// TIA Portal V17 export
// export: Created 2025-03-07T09:17:48.5611962Z, ExportSetting WithDefaults, DisplayName Totally Integrated Automation Portal, DisplayVersion V17 Update 8, DisplayName TIA Portal Openness, DisplayVersion V17 Update 8, DisplayName TIA Portal Version Control Interface, DisplayVersion V17, DisplayName SINAMICS Startdrive Advanced, DisplayVersion V17 SP2, DisplayName SINAMICS Startdrive G110M, G120, G120C, G120D, G120P, G115D, DisplayVersion V17 SP2, DisplayName SINAMICS Startdrive G130, G150, S120, S150, SINAMICS MV, S210, DisplayVersion V17 SP2, DisplayName STEP 7 Professional, DisplayVersion V17 Update 8, DisplayName SINUMERIK ONE STEP 7 Toolbox, DisplayVersion V17 Update 12, DisplayName SINUMERIK 840D sl STEP 7 Toolbox, DisplayVersion V17 Update 12, DisplayName STEP 7 Safety, DisplayVersion V17 Update 6, DisplayName WinCC Advanced, DisplayVersion V17 Update 8
FUNCTION "FC2102_INFEED_MODULE" : Void   // FC2102, LAD
{ S7_Optimized_Access := 'FALSE' }
AUTHOR : ETXETAR
VERSION : 1.0
// stored: AutoNumber false, IsIECCheckEnabled false, SetENOAutomatically false, UDAEnableTagReadback false
   VAR_TEMP
      O_BYTE_0 : Struct   // OPTIONS BYTE 0
         POWER_SUPPLY_2 : Bool;   // POWER SUPPLY 2 OPTION
      END_STRUCT;
   END_VAR
   VAR CONSTANT
      FC_NUMBER : DInt := 2102;
   END_VAR
   VAR_TEMP   // added for the SCL form of the ladder/FBD networks
      _w1 : Bool;
   END_VAR
BEGIN

REGION Network 1: OPTIONS OFF
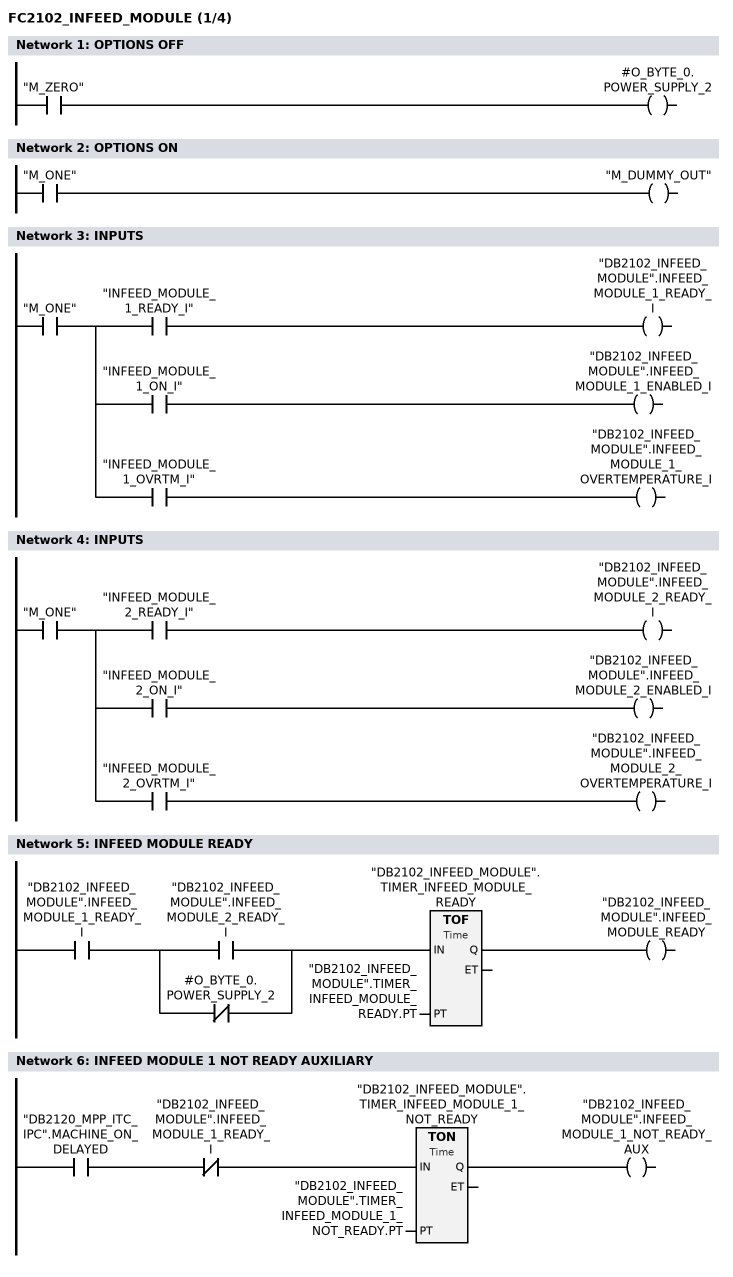
   RUNG wire#powerrail
      Contact( "M_ZERO" )
      Coil( #O_BYTE_0.POWER_SUPPLY_2 )
   END_RUNG
   // the same network as SCL:
   #O_BYTE_0.POWER_SUPPLY_2 := "M_ZERO";
END_REGION

REGION Network 2: OPTIONS ON
   RUNG wire#powerrail
      Contact( "M_ONE" )
      Coil( "M_DUMMY_OUT" )
   END_RUNG
   // the same network as SCL:
   "M_DUMMY_OUT" := "M_ONE";
END_REGION

REGION Network 3: INPUTS
   RUNG wire#powerrail
      Contact( "M_ONE" )
      wire#w1
      Contact( "INFEED_MODULE_1_READY_I" )
      Coil( "DB2102_INFEED_MODULE".INFEED_MODULE_1_READY_I )
   END_RUNG
   RUNG wire#w1
      Contact( "INFEED_MODULE_1_ON_I" )
      Coil( "DB2102_INFEED_MODULE".INFEED_MODULE_1_ENABLED_I )
   END_RUNG
   RUNG wire#w1
      Contact( "INFEED_MODULE_1_OVRTM_I" )
      Coil( "DB2102_INFEED_MODULE".INFEED_MODULE_1_OVERTEMPERATURE_I )
   END_RUNG
   // the same network as SCL:
   "DB2102_INFEED_MODULE".INFEED_MODULE_1_READY_I := "M_ONE" AND "INFEED_MODULE_1_READY_I";
   "DB2102_INFEED_MODULE".INFEED_MODULE_1_ENABLED_I := "M_ONE" AND "INFEED_MODULE_1_ON_I";
   "DB2102_INFEED_MODULE".INFEED_MODULE_1_OVERTEMPERATURE_I := "M_ONE" AND "INFEED_MODULE_1_OVRTM_I";
END_REGION

REGION Network 4: INPUTS
   RUNG wire#powerrail
      Contact( "M_ONE" )
      wire#w1
      Contact( "INFEED_MODULE_2_READY_I" )
      Coil( "DB2102_INFEED_MODULE".INFEED_MODULE_2_READY_I )
   END_RUNG
   RUNG wire#w1
      Contact( "INFEED_MODULE_2_ON_I" )
      Coil( "DB2102_INFEED_MODULE".INFEED_MODULE_2_ENABLED_I )
   END_RUNG
   RUNG wire#w1
      Contact( "INFEED_MODULE_2_OVRTM_I" )
      Coil( "DB2102_INFEED_MODULE".INFEED_MODULE_2_OVERTEMPERATURE_I )
   END_RUNG
   // the same network as SCL:
   "DB2102_INFEED_MODULE".INFEED_MODULE_2_READY_I := "M_ONE" AND "INFEED_MODULE_2_READY_I";
   "DB2102_INFEED_MODULE".INFEED_MODULE_2_ENABLED_I := "M_ONE" AND "INFEED_MODULE_2_ON_I";
   "DB2102_INFEED_MODULE".INFEED_MODULE_2_OVERTEMPERATURE_I := "M_ONE" AND "INFEED_MODULE_2_OVRTM_I";
END_REGION

REGION Network 5: INFEED MODULE READY
   RUNG wire#powerrail
      Contact( "DB2102_INFEED_MODULE".INFEED_MODULE_1_READY_I )
      wire#w1
      Contact( "DB2102_INFEED_MODULE".INFEED_MODULE_2_READY_I )
      wire#w2
      { S7_Templates := "time_type := Time" } "DB2102_INFEED_MODULE".TIMER_INFEED_MODULE_READY.TOF(pt := "DB2102_INFEED_MODULE".TIMER_INFEED_MODULE_READY.PT, et =>)
      Coil( "DB2102_INFEED_MODULE".INFEED_MODULE_READY )
   END_RUNG
   RUNG wire#w1
      I_Contact( #O_BYTE_0.POWER_SUPPLY_2 )
   END_RUNG wire#w2
   // the same network as SCL:
   "DB2102_INFEED_MODULE".TIMER_INFEED_MODULE_READY.TOF(IN := "DB2102_INFEED_MODULE".INFEED_MODULE_1_READY_I AND ("DB2102_INFEED_MODULE".INFEED_MODULE_2_READY_I OR NOT #O_BYTE_0.POWER_SUPPLY_2),
                           PT := "DB2102_INFEED_MODULE".TIMER_INFEED_MODULE_READY.PT);
   "DB2102_INFEED_MODULE".INFEED_MODULE_READY := "DB2102_INFEED_MODULE".TIMER_INFEED_MODULE_READY.Q;
END_REGION

REGION Network 6: INFEED MODULE 1 NOT READY AUXILIARY
   RUNG wire#powerrail
      Contact( "DB2120_MPP_ITC_IPC".MACHINE_ON_DELAYED )
      I_Contact( "DB2102_INFEED_MODULE".INFEED_MODULE_1_READY_I )
      { S7_Templates := "time_type := Time" } "DB2102_INFEED_MODULE".TIMER_INFEED_MODULE_1_NOT_READY.TON(pt := "DB2102_INFEED_MODULE".TIMER_INFEED_MODULE_1_NOT_READY.PT, et =>)
      Coil( "DB2102_INFEED_MODULE".INFEED_MODULE_1_NOT_READY_AUX )
   END_RUNG
   // the same network as SCL:
   "DB2102_INFEED_MODULE".TIMER_INFEED_MODULE_1_NOT_READY.TON(IN := "DB2120_MPP_ITC_IPC".MACHINE_ON_DELAYED AND NOT "DB2102_INFEED_MODULE".INFEED_MODULE_1_READY_I,
                           PT := "DB2102_INFEED_MODULE".TIMER_INFEED_MODULE_1_NOT_READY.PT);
   "DB2102_INFEED_MODULE".INFEED_MODULE_1_NOT_READY_AUX := "DB2102_INFEED_MODULE".TIMER_INFEED_MODULE_1_NOT_READY.Q;
END_REGION

REGION Network 7: INFEED MODULE 1 NOT READY ALARM
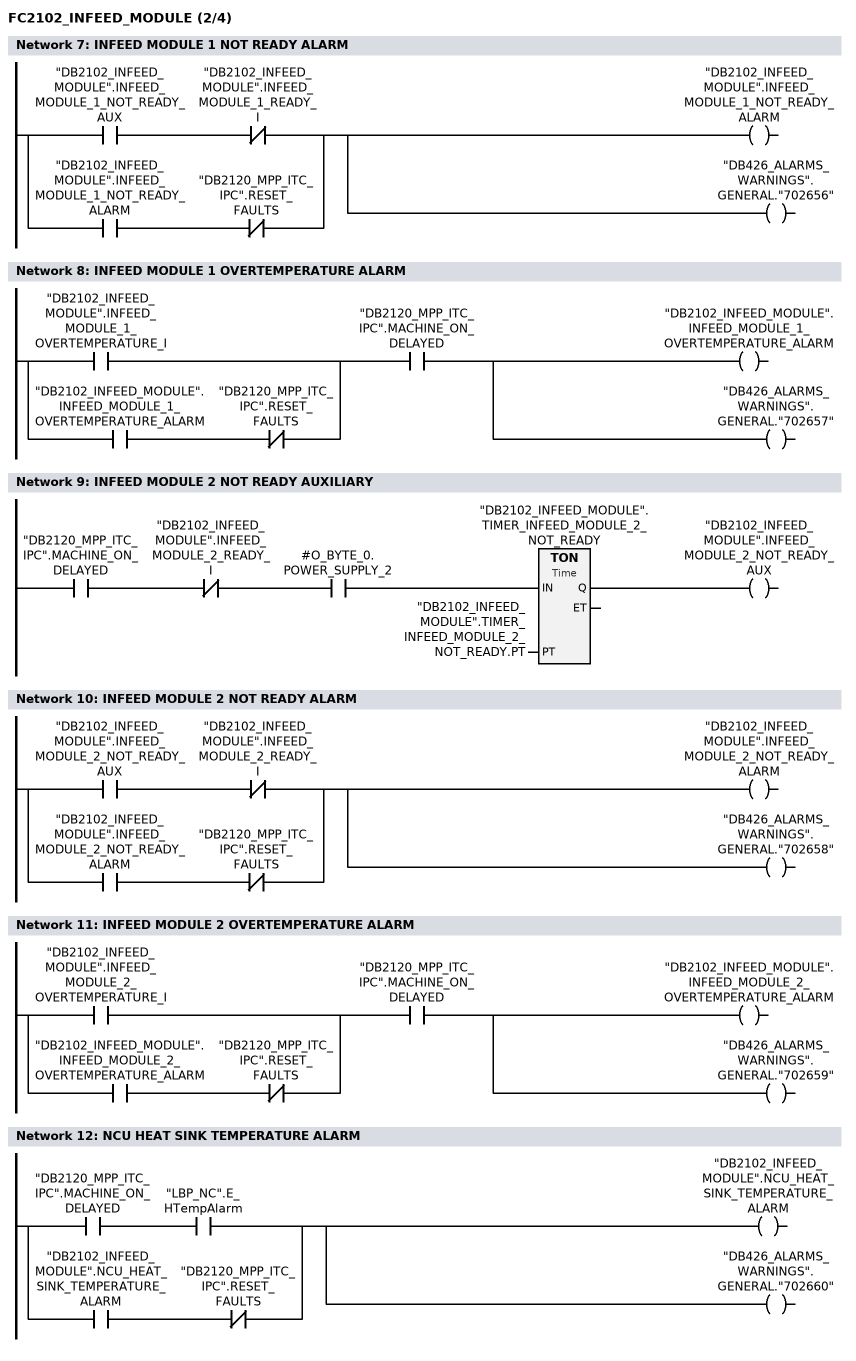
   RUNG wire#powerrail
      Contact( "DB2102_INFEED_MODULE".INFEED_MODULE_1_NOT_READY_AUX )
      I_Contact( "DB2102_INFEED_MODULE".INFEED_MODULE_1_READY_I )
      wire#w1
      Coil( "DB2102_INFEED_MODULE".INFEED_MODULE_1_NOT_READY_ALARM )
   END_RUNG
   RUNG wire#powerrail
      Contact( "DB2102_INFEED_MODULE".INFEED_MODULE_1_NOT_READY_ALARM )
      I_Contact( "DB2120_MPP_ITC_IPC".RESET_FAULTS )
   END_RUNG wire#w1
   RUNG wire#w1
      Coil( "DB426_ALARMS_WARNINGS".GENERAL."702656" )
   END_RUNG
   // the same network as SCL:
   "DB2102_INFEED_MODULE".INFEED_MODULE_1_NOT_READY_ALARM := ("DB2102_INFEED_MODULE".INFEED_MODULE_1_NOT_READY_AUX AND NOT "DB2102_INFEED_MODULE".INFEED_MODULE_1_READY_I) OR ("DB2102_INFEED_MODULE".INFEED_MODULE_1_NOT_READY_ALARM AND NOT "DB2120_MPP_ITC_IPC".RESET_FAULTS);
   "DB426_ALARMS_WARNINGS".GENERAL."702656" := "DB2102_INFEED_MODULE".INFEED_MODULE_1_NOT_READY_ALARM;
END_REGION

REGION Network 8: INFEED MODULE 1 OVERTEMPERATURE ALARM
   RUNG wire#powerrail
      Contact( "DB2102_INFEED_MODULE".INFEED_MODULE_1_OVERTEMPERATURE_I )
      wire#w1
      Contact( "DB2120_MPP_ITC_IPC".MACHINE_ON_DELAYED )
      wire#w2
      Coil( "DB2102_INFEED_MODULE".INFEED_MODULE_1_OVERTEMPERATURE_ALARM )
   END_RUNG
   RUNG wire#powerrail
      Contact( "DB2102_INFEED_MODULE".INFEED_MODULE_1_OVERTEMPERATURE_ALARM )
      I_Contact( "DB2120_MPP_ITC_IPC".RESET_FAULTS )
   END_RUNG wire#w1
   RUNG wire#w2
      Coil( "DB426_ALARMS_WARNINGS".GENERAL."702657" )
   END_RUNG
   // the same network as SCL:
   "DB2102_INFEED_MODULE".INFEED_MODULE_1_OVERTEMPERATURE_ALARM := ("DB2102_INFEED_MODULE".INFEED_MODULE_1_OVERTEMPERATURE_I OR ("DB2102_INFEED_MODULE".INFEED_MODULE_1_OVERTEMPERATURE_ALARM AND NOT "DB2120_MPP_ITC_IPC".RESET_FAULTS)) AND "DB2120_MPP_ITC_IPC".MACHINE_ON_DELAYED;
   "DB426_ALARMS_WARNINGS".GENERAL."702657" := "DB2102_INFEED_MODULE".INFEED_MODULE_1_OVERTEMPERATURE_ALARM;
END_REGION

REGION Network 9: INFEED MODULE 2 NOT READY AUXILIARY
   RUNG wire#powerrail
      Contact( "DB2120_MPP_ITC_IPC".MACHINE_ON_DELAYED )
      I_Contact( "DB2102_INFEED_MODULE".INFEED_MODULE_2_READY_I )
      Contact( #O_BYTE_0.POWER_SUPPLY_2 )
      { S7_Templates := "time_type := Time" } "DB2102_INFEED_MODULE".TIMER_INFEED_MODULE_2_NOT_READY.TON(pt := "DB2102_INFEED_MODULE".TIMER_INFEED_MODULE_2_NOT_READY.PT, et =>)
      Coil( "DB2102_INFEED_MODULE".INFEED_MODULE_2_NOT_READY_AUX )
   END_RUNG
   // the same network as SCL:
   "DB2102_INFEED_MODULE".TIMER_INFEED_MODULE_2_NOT_READY.TON(IN := "DB2120_MPP_ITC_IPC".MACHINE_ON_DELAYED AND NOT "DB2102_INFEED_MODULE".INFEED_MODULE_2_READY_I AND #O_BYTE_0.POWER_SUPPLY_2,
                           PT := "DB2102_INFEED_MODULE".TIMER_INFEED_MODULE_2_NOT_READY.PT);
   "DB2102_INFEED_MODULE".INFEED_MODULE_2_NOT_READY_AUX := "DB2102_INFEED_MODULE".TIMER_INFEED_MODULE_2_NOT_READY.Q;
END_REGION

REGION Network 10: INFEED MODULE 2 NOT READY ALARM
   RUNG wire#powerrail
      Contact( "DB2102_INFEED_MODULE".INFEED_MODULE_2_NOT_READY_AUX )
      I_Contact( "DB2102_INFEED_MODULE".INFEED_MODULE_2_READY_I )
      wire#w1
      Coil( "DB2102_INFEED_MODULE".INFEED_MODULE_2_NOT_READY_ALARM )
   END_RUNG
   RUNG wire#powerrail
      Contact( "DB2102_INFEED_MODULE".INFEED_MODULE_2_NOT_READY_ALARM )
      I_Contact( "DB2120_MPP_ITC_IPC".RESET_FAULTS )
   END_RUNG wire#w1
   RUNG wire#w1
      Coil( "DB426_ALARMS_WARNINGS".GENERAL."702658" )
   END_RUNG
   // the same network as SCL:
   "DB2102_INFEED_MODULE".INFEED_MODULE_2_NOT_READY_ALARM := ("DB2102_INFEED_MODULE".INFEED_MODULE_2_NOT_READY_AUX AND NOT "DB2102_INFEED_MODULE".INFEED_MODULE_2_READY_I) OR ("DB2102_INFEED_MODULE".INFEED_MODULE_2_NOT_READY_ALARM AND NOT "DB2120_MPP_ITC_IPC".RESET_FAULTS);
   "DB426_ALARMS_WARNINGS".GENERAL."702658" := "DB2102_INFEED_MODULE".INFEED_MODULE_2_NOT_READY_ALARM;
END_REGION

REGION Network 11: INFEED MODULE 2 OVERTEMPERATURE ALARM
   RUNG wire#powerrail
      Contact( "DB2102_INFEED_MODULE".INFEED_MODULE_2_OVERTEMPERATURE_I )
      wire#w1
      Contact( "DB2120_MPP_ITC_IPC".MACHINE_ON_DELAYED )
      wire#w2
      Coil( "DB2102_INFEED_MODULE".INFEED_MODULE_2_OVERTEMPERATURE_ALARM )
   END_RUNG
   RUNG wire#powerrail
      Contact( "DB2102_INFEED_MODULE".INFEED_MODULE_2_OVERTEMPERATURE_ALARM )
      I_Contact( "DB2120_MPP_ITC_IPC".RESET_FAULTS )
   END_RUNG wire#w1
   RUNG wire#w2
      Coil( "DB426_ALARMS_WARNINGS".GENERAL."702659" )
   END_RUNG
   // the same network as SCL:
   "DB2102_INFEED_MODULE".INFEED_MODULE_2_OVERTEMPERATURE_ALARM := ("DB2102_INFEED_MODULE".INFEED_MODULE_2_OVERTEMPERATURE_I OR ("DB2102_INFEED_MODULE".INFEED_MODULE_2_OVERTEMPERATURE_ALARM AND NOT "DB2120_MPP_ITC_IPC".RESET_FAULTS)) AND "DB2120_MPP_ITC_IPC".MACHINE_ON_DELAYED;
   "DB426_ALARMS_WARNINGS".GENERAL."702659" := "DB2102_INFEED_MODULE".INFEED_MODULE_2_OVERTEMPERATURE_ALARM;
END_REGION

REGION Network 12: NCU HEAT SINK TEMPERATURE ALARM
   RUNG wire#powerrail
      Contact( "DB2120_MPP_ITC_IPC".MACHINE_ON_DELAYED )
      Contact( "LBP_NC".E_HTempAlarm )
      wire#w1
      Coil( "DB2102_INFEED_MODULE".NCU_HEAT_SINK_TEMPERATURE_ALARM )
   END_RUNG
   RUNG wire#powerrail
      Contact( "DB2102_INFEED_MODULE".NCU_HEAT_SINK_TEMPERATURE_ALARM )
      I_Contact( "DB2120_MPP_ITC_IPC".RESET_FAULTS )
   END_RUNG wire#w1
   RUNG wire#w1
      Coil( "DB426_ALARMS_WARNINGS".GENERAL."702660" )
   END_RUNG
   // the same network as SCL:
   "DB2102_INFEED_MODULE".NCU_HEAT_SINK_TEMPERATURE_ALARM := ("DB2120_MPP_ITC_IPC".MACHINE_ON_DELAYED AND "LBP_NC".E_HTempAlarm) OR ("DB2102_INFEED_MODULE".NCU_HEAT_SINK_TEMPERATURE_ALARM AND NOT "DB2120_MPP_ITC_IPC".RESET_FAULTS);
   "DB426_ALARMS_WARNINGS".GENERAL."702660" := "DB2102_INFEED_MODULE".NCU_HEAT_SINK_TEMPERATURE_ALARM;
END_REGION

REGION Network 13: NCU LOW BATTERY ALARM
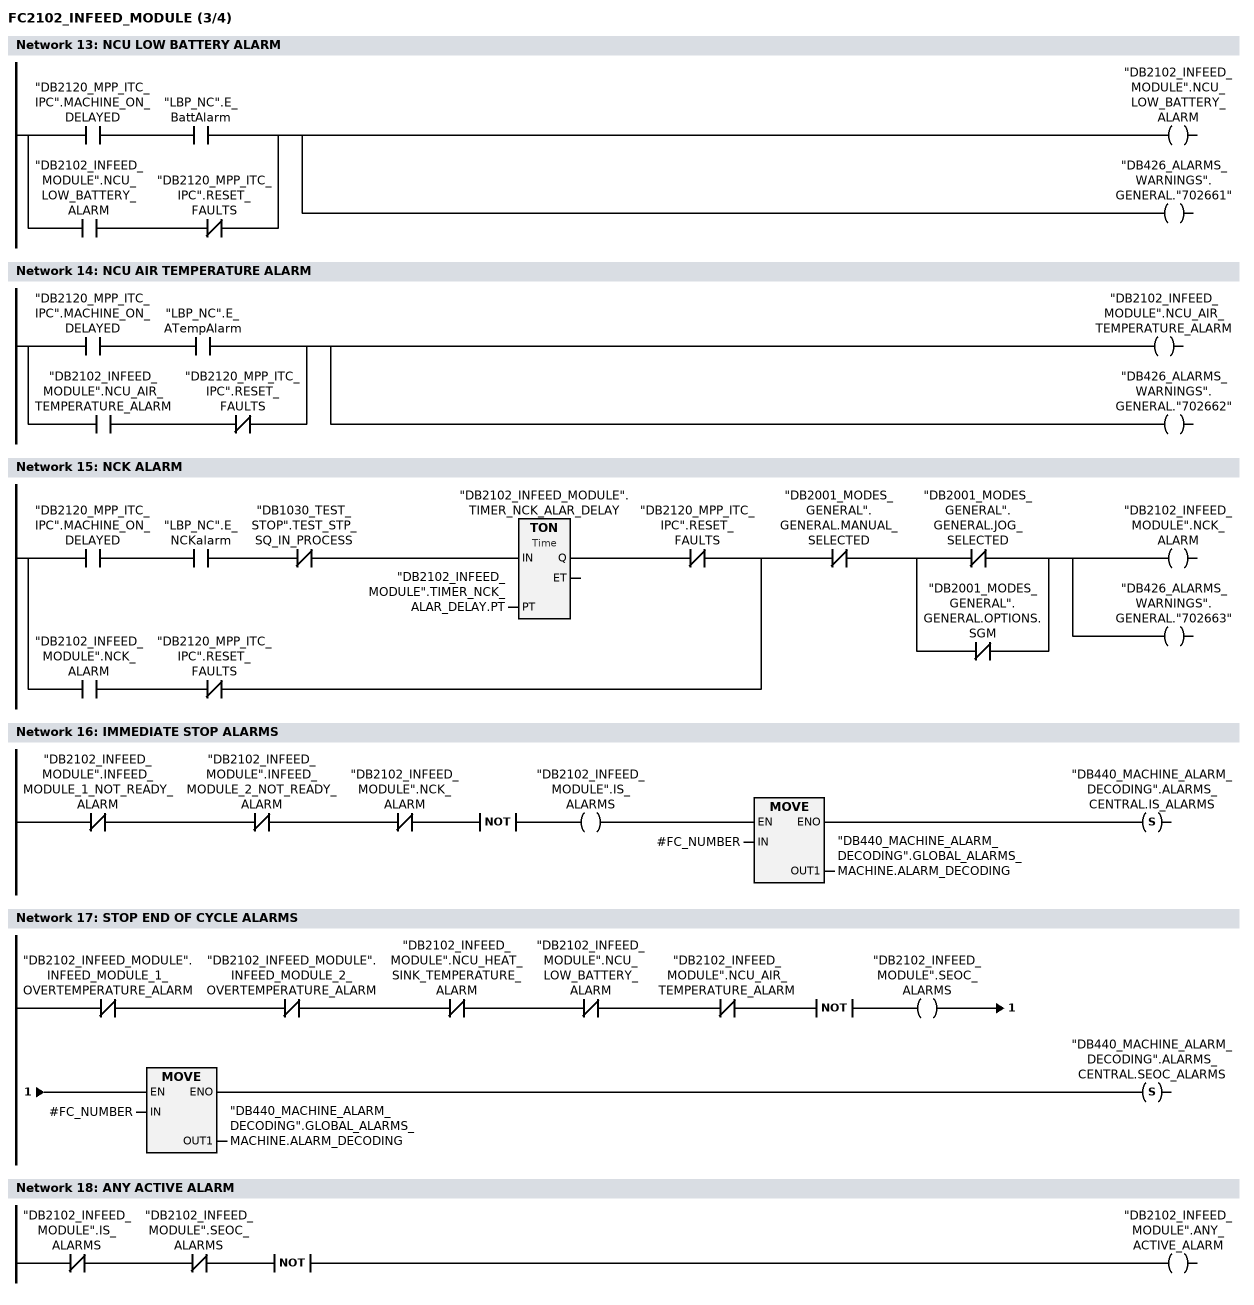
   RUNG wire#powerrail
      Contact( "DB2120_MPP_ITC_IPC".MACHINE_ON_DELAYED )
      Contact( "LBP_NC".E_BattAlarm )
      wire#w1
      Coil( "DB2102_INFEED_MODULE".NCU_LOW_BATTERY_ALARM )
   END_RUNG
   RUNG wire#powerrail
      Contact( "DB2102_INFEED_MODULE".NCU_LOW_BATTERY_ALARM )
      I_Contact( "DB2120_MPP_ITC_IPC".RESET_FAULTS )
   END_RUNG wire#w1
   RUNG wire#w1
      Coil( "DB426_ALARMS_WARNINGS".GENERAL."702661" )
   END_RUNG
   // the same network as SCL:
   "DB2102_INFEED_MODULE".NCU_LOW_BATTERY_ALARM := ("DB2120_MPP_ITC_IPC".MACHINE_ON_DELAYED AND "LBP_NC".E_BattAlarm) OR ("DB2102_INFEED_MODULE".NCU_LOW_BATTERY_ALARM AND NOT "DB2120_MPP_ITC_IPC".RESET_FAULTS);
   "DB426_ALARMS_WARNINGS".GENERAL."702661" := "DB2102_INFEED_MODULE".NCU_LOW_BATTERY_ALARM;
END_REGION

REGION Network 14: NCU AIR TEMPERATURE ALARM
   RUNG wire#powerrail
      Contact( "DB2120_MPP_ITC_IPC".MACHINE_ON_DELAYED )
      Contact( "LBP_NC".E_ATempAlarm )
      wire#w1
      Coil( "DB2102_INFEED_MODULE".NCU_AIR_TEMPERATURE_ALARM )
   END_RUNG
   RUNG wire#powerrail
      Contact( "DB2102_INFEED_MODULE".NCU_AIR_TEMPERATURE_ALARM )
      I_Contact( "DB2120_MPP_ITC_IPC".RESET_FAULTS )
   END_RUNG wire#w1
   RUNG wire#w1
      Coil( "DB426_ALARMS_WARNINGS".GENERAL."702662" )
   END_RUNG
   // the same network as SCL:
   "DB2102_INFEED_MODULE".NCU_AIR_TEMPERATURE_ALARM := ("DB2120_MPP_ITC_IPC".MACHINE_ON_DELAYED AND "LBP_NC".E_ATempAlarm) OR ("DB2102_INFEED_MODULE".NCU_AIR_TEMPERATURE_ALARM AND NOT "DB2120_MPP_ITC_IPC".RESET_FAULTS);
   "DB426_ALARMS_WARNINGS".GENERAL."702662" := "DB2102_INFEED_MODULE".NCU_AIR_TEMPERATURE_ALARM;
END_REGION

REGION Network 15: NCK ALARM
   RUNG wire#powerrail
      Contact( "DB2120_MPP_ITC_IPC".MACHINE_ON_DELAYED )
      Contact( "LBP_NC".E_NCKalarm )
      I_Contact( "DB1030_TEST_STOP".TEST_STP_SQ_IN_PROCESS )
      { S7_Templates := "time_type := Time" } "DB2102_INFEED_MODULE".TIMER_NCK_ALAR_DELAY.TON(pt := "DB2102_INFEED_MODULE".TIMER_NCK_ALAR_DELAY.PT, et =>)
      I_Contact( "DB2120_MPP_ITC_IPC".RESET_FAULTS )
      wire#w1
      I_Contact( "DB2001_MODES_GENERAL".GENERAL.MANUAL_SELECTED )
      wire#w2
      I_Contact( "DB2001_MODES_GENERAL".GENERAL.JOG_SELECTED )
      wire#w3
      Coil( "DB2102_INFEED_MODULE".NCK_ALARM )
   END_RUNG
   RUNG wire#powerrail
      Contact( "DB2102_INFEED_MODULE".NCK_ALARM )
      I_Contact( "DB2120_MPP_ITC_IPC".RESET_FAULTS )
   END_RUNG wire#w1
   RUNG wire#w2
      I_Contact( "DB2001_MODES_GENERAL".GENERAL.OPTIONS.SGM )
   END_RUNG wire#w3
   RUNG wire#w3
      Coil( "DB426_ALARMS_WARNINGS".GENERAL."702663" )
   END_RUNG
   // the same network as SCL:
   "DB2102_INFEED_MODULE".TIMER_NCK_ALAR_DELAY.TON(IN := "DB2120_MPP_ITC_IPC".MACHINE_ON_DELAYED AND "LBP_NC".E_NCKalarm AND NOT "DB1030_TEST_STOP".TEST_STP_SQ_IN_PROCESS,
                           PT := "DB2102_INFEED_MODULE".TIMER_NCK_ALAR_DELAY.PT);
   "DB2102_INFEED_MODULE".NCK_ALARM := (("DB2102_INFEED_MODULE".TIMER_NCK_ALAR_DELAY.Q AND NOT "DB2120_MPP_ITC_IPC".RESET_FAULTS) OR ("DB2102_INFEED_MODULE".NCK_ALARM AND NOT "DB2120_MPP_ITC_IPC".RESET_FAULTS)) AND NOT "DB2001_MODES_GENERAL".GENERAL.MANUAL_SELECTED AND (NOT "DB2001_MODES_GENERAL".GENERAL.JOG_SELECTED OR NOT "DB2001_MODES_GENERAL".GENERAL.OPTIONS.SGM);
   "DB426_ALARMS_WARNINGS".GENERAL."702663" := "DB2102_INFEED_MODULE".NCK_ALARM;
END_REGION

REGION Network 16: IMMEDIATE STOP ALARMS
   RUNG wire#powerrail
      I_Contact( "DB2102_INFEED_MODULE".INFEED_MODULE_1_NOT_READY_ALARM )
      I_Contact( "DB2102_INFEED_MODULE".INFEED_MODULE_2_NOT_READY_ALARM )
      I_Contact( "DB2102_INFEED_MODULE".NCK_ALARM )
      Not()
      Coil( "DB2102_INFEED_MODULE".IS_ALARMS )
      { S7_GenerateENO := "TRUE" } Move(in := #FC_NUMBER, out1 => "DB440_MACHINE_ALARM_DECODING".GLOBAL_ALARMS_MACHINE.ALARM_DECODING)
      S_Coil( "DB440_MACHINE_ALARM_DECODING".ALARMS_CENTRAL.IS_ALARMS )
   END_RUNG
   // the same network as SCL:
   // ENO of a box is taken as its EN; it also drops when the box reports an error
   "DB2102_INFEED_MODULE".IS_ALARMS := NOT (NOT "DB2102_INFEED_MODULE".INFEED_MODULE_1_NOT_READY_ALARM AND NOT "DB2102_INFEED_MODULE".INFEED_MODULE_2_NOT_READY_ALARM AND NOT "DB2102_INFEED_MODULE".NCK_ALARM);
   IF "DB2102_INFEED_MODULE".IS_ALARMS THEN
       "DB440_MACHINE_ALARM_DECODING".GLOBAL_ALARMS_MACHINE.ALARM_DECODING := #FC_NUMBER;
       "DB440_MACHINE_ALARM_DECODING".ALARMS_CENTRAL.IS_ALARMS := TRUE;
   END_IF;
END_REGION

REGION Network 17: STOP END OF CYCLE ALARMS
   RUNG wire#powerrail
      I_Contact( "DB2102_INFEED_MODULE".INFEED_MODULE_1_OVERTEMPERATURE_ALARM )
      I_Contact( "DB2102_INFEED_MODULE".INFEED_MODULE_2_OVERTEMPERATURE_ALARM )
      I_Contact( "DB2102_INFEED_MODULE".NCU_HEAT_SINK_TEMPERATURE_ALARM )
      I_Contact( "DB2102_INFEED_MODULE".NCU_LOW_BATTERY_ALARM )
      I_Contact( "DB2102_INFEED_MODULE".NCU_AIR_TEMPERATURE_ALARM )
      Not()
      Coil( "DB2102_INFEED_MODULE".SEOC_ALARMS )
      { S7_GenerateENO := "TRUE" } Move(in := #FC_NUMBER, out1 => "DB440_MACHINE_ALARM_DECODING".GLOBAL_ALARMS_MACHINE.ALARM_DECODING)
      S_Coil( "DB440_MACHINE_ALARM_DECODING".ALARMS_CENTRAL.SEOC_ALARMS )
   END_RUNG
   // the same network as SCL:
   // ENO of a box is taken as its EN; it also drops when the box reports an error
   "DB2102_INFEED_MODULE".SEOC_ALARMS := NOT (NOT "DB2102_INFEED_MODULE".INFEED_MODULE_1_OVERTEMPERATURE_ALARM AND NOT "DB2102_INFEED_MODULE".INFEED_MODULE_2_OVERTEMPERATURE_ALARM AND NOT "DB2102_INFEED_MODULE".NCU_HEAT_SINK_TEMPERATURE_ALARM AND NOT "DB2102_INFEED_MODULE".NCU_LOW_BATTERY_ALARM AND NOT "DB2102_INFEED_MODULE".NCU_AIR_TEMPERATURE_ALARM);
   IF "DB2102_INFEED_MODULE".SEOC_ALARMS THEN
       "DB440_MACHINE_ALARM_DECODING".GLOBAL_ALARMS_MACHINE.ALARM_DECODING := #FC_NUMBER;
       "DB440_MACHINE_ALARM_DECODING".ALARMS_CENTRAL.SEOC_ALARMS := TRUE;
   END_IF;
END_REGION

REGION Network 18: ANY ACTIVE ALARM
   RUNG wire#powerrail
      I_Contact( "DB2102_INFEED_MODULE".IS_ALARMS )
      I_Contact( "DB2102_INFEED_MODULE".SEOC_ALARMS )
      Not()
      Coil( "DB2102_INFEED_MODULE".ANY_ACTIVE_ALARM )
   END_RUNG
   // the same network as SCL:
   "DB2102_INFEED_MODULE".ANY_ACTIVE_ALARM := NOT (NOT "DB2102_INFEED_MODULE".IS_ALARMS AND NOT "DB2102_INFEED_MODULE".SEOC_ALARMS);
END_REGION

REGION Network 19: INFEED MODULE OFF 3 OUTPUT
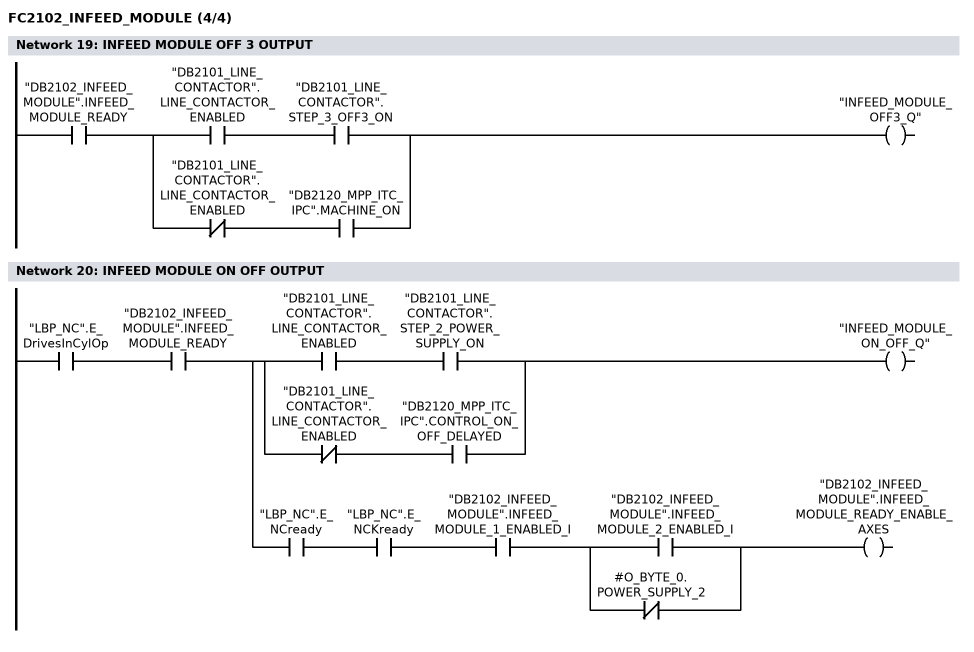
   RUNG wire#powerrail
      Contact( "DB2102_INFEED_MODULE".INFEED_MODULE_READY )
      wire#w1
      Contact( "DB2101_LINE_CONTACTOR".LINE_CONTACTOR_ENABLED )
      Contact( "DB2101_LINE_CONTACTOR".STEP_3_OFF3_ON )
      wire#w2
      Coil( "INFEED_MODULE_OFF3_Q" )
   END_RUNG
   RUNG wire#w1
      I_Contact( "DB2101_LINE_CONTACTOR".LINE_CONTACTOR_ENABLED )
      Contact( "DB2120_MPP_ITC_IPC".MACHINE_ON )
   END_RUNG wire#w2
   // the same network as SCL:
   "INFEED_MODULE_OFF3_Q" := "DB2102_INFEED_MODULE".INFEED_MODULE_READY AND (("DB2101_LINE_CONTACTOR".LINE_CONTACTOR_ENABLED AND "DB2101_LINE_CONTACTOR".STEP_3_OFF3_ON) OR (NOT "DB2101_LINE_CONTACTOR".LINE_CONTACTOR_ENABLED AND "DB2120_MPP_ITC_IPC".MACHINE_ON));
END_REGION

REGION Network 20: INFEED MODULE ON OFF OUTPUT
   RUNG wire#powerrail
      Contact( "LBP_NC".E_DrivesInCylOp )
      Contact( "DB2102_INFEED_MODULE".INFEED_MODULE_READY )
      wire#w1
      Contact( "DB2101_LINE_CONTACTOR".LINE_CONTACTOR_ENABLED )
      Contact( "DB2101_LINE_CONTACTOR".STEP_2_POWER_SUPPLY_ON )
      wire#w2
      Coil( "INFEED_MODULE_ON_OFF_Q" )
   END_RUNG
   RUNG wire#w1
      I_Contact( "DB2101_LINE_CONTACTOR".LINE_CONTACTOR_ENABLED )
      Contact( "DB2120_MPP_ITC_IPC".CONTROL_ON_OFF_DELAYED )
   END_RUNG wire#w2
   RUNG wire#w1
      Contact( "LBP_NC".E_NCready )
      Contact( "LBP_NC".E_NCKready )
      Contact( "DB2102_INFEED_MODULE".INFEED_MODULE_1_ENABLED_I )
      wire#w3
      Contact( "DB2102_INFEED_MODULE".INFEED_MODULE_2_ENABLED_I )
      wire#w4
      Coil( "DB2102_INFEED_MODULE".INFEED_MODULE_READY_ENABLE_AXES )
   END_RUNG
   RUNG wire#w3
      I_Contact( #O_BYTE_0.POWER_SUPPLY_2 )
   END_RUNG wire#w4
   // the same network as SCL:
   #_w1 := "LBP_NC".E_DrivesInCylOp AND "DB2102_INFEED_MODULE".INFEED_MODULE_READY;
   "INFEED_MODULE_ON_OFF_Q" := #_w1 AND (("DB2101_LINE_CONTACTOR".LINE_CONTACTOR_ENABLED AND "DB2101_LINE_CONTACTOR".STEP_2_POWER_SUPPLY_ON) OR (NOT "DB2101_LINE_CONTACTOR".LINE_CONTACTOR_ENABLED AND "DB2120_MPP_ITC_IPC".CONTROL_ON_OFF_DELAYED));
   "DB2102_INFEED_MODULE".INFEED_MODULE_READY_ENABLE_AXES := #_w1 AND "LBP_NC".E_NCready AND "LBP_NC".E_NCKready AND "DB2102_INFEED_MODULE".INFEED_MODULE_1_ENABLED_I AND ("DB2102_INFEED_MODULE".INFEED_MODULE_2_ENABLED_I OR NOT #O_BYTE_0.POWER_SUPPLY_2);
END_REGION
END_FUNCTION
